// TIA Portal V21 export
FUNCTION "DELTA" : Void   // FC18, LAD
{ S7_Optimized_Access := 'TRUE' }
// stored: SetENOAutomatically false
   VAR_TEMP
      "F1 VALUE" : Real;
      "F2 VALUE" : Real;
      "F3 VALUE" : Real;
      "F4 VALUE" : Real;
      "F5 VALUE" : Real;
   END_VAR
   VAR_TEMP   // added for the SCL form of the ladder/FBD networks
      _w1 : Bool;
      _w2 : Bool;
      _w3 : Bool;
      _w4 : Bool;
      _w5 : Bool;
      _w6 : Bool;
      _w7 : Bool;
      _w8 : Bool;
      _w9 : Bool;
      _w10 : Bool;
      _w11 : Bool;
      _w12 : Bool;
   END_VAR
BEGIN

REGION Network 1
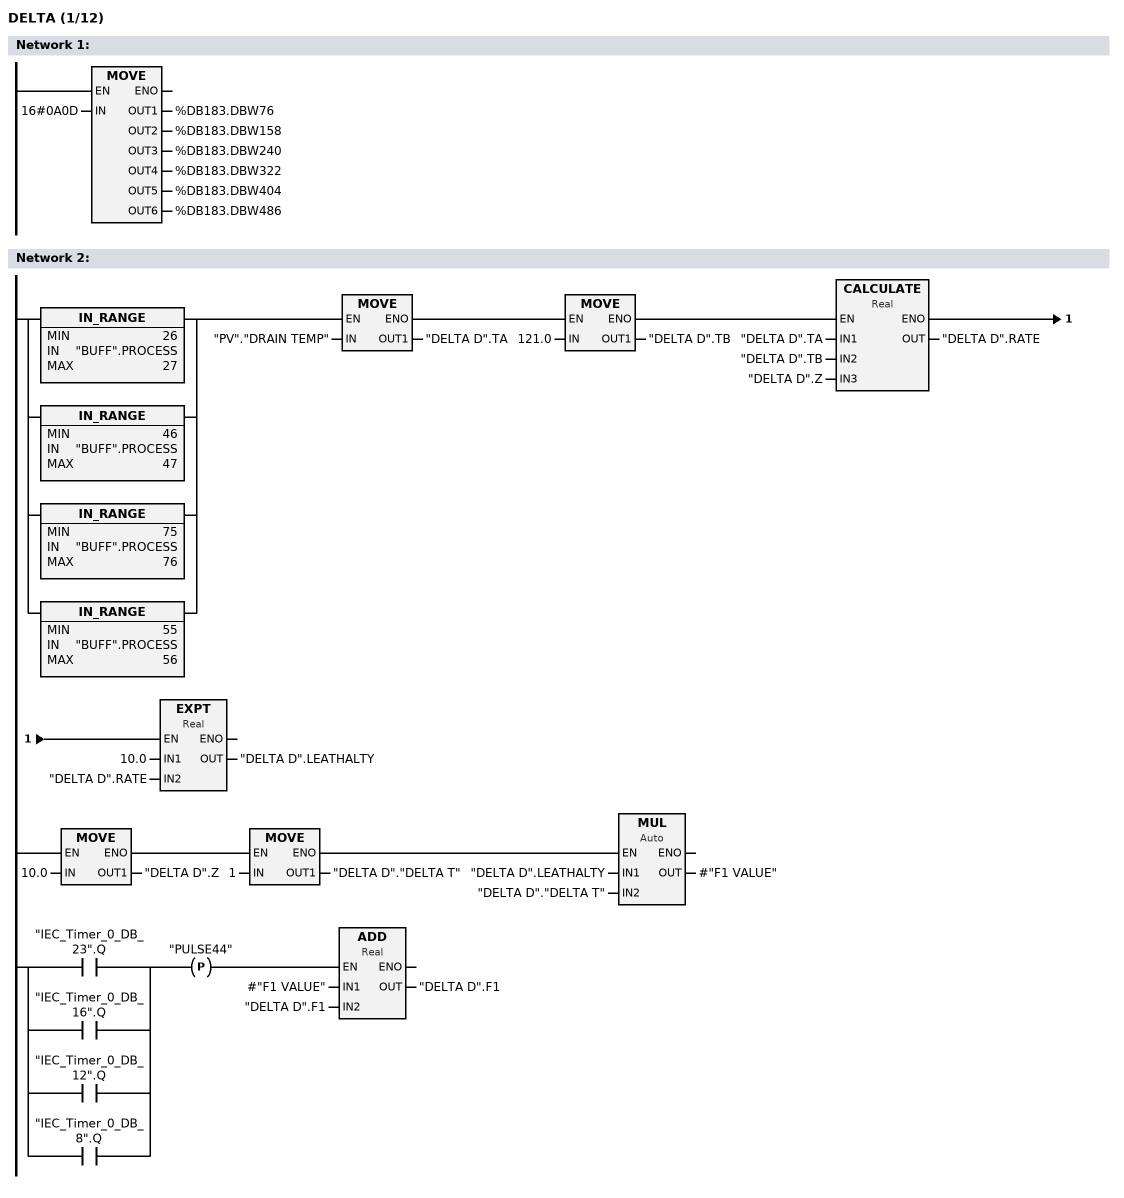
   RUNG wire#powerrail
      Move(in := 16#0A0D, out1 => %DB183.DBW76, out2 => %DB183.DBW158, out3 => %DB183.DBW240, out4 => %DB183.DBW322, out5 => %DB183.DBW404, out6 => %DB183.DBW486)
   END_RUNG
   // the same network as SCL:
   %DB183.DBW76 := 16#0A0D;
   %DB183.DBW158 := 16#0A0D;
   %DB183.DBW240 := 16#0A0D;
   %DB183.DBW322 := 16#0A0D;
   %DB183.DBW404 := 16#0A0D;
   %DB183.DBW486 := 16#0A0D;
END_REGION

REGION Network 2
   IF ((26 <= "BUFF".PROCESS) AND ("BUFF".PROCESS <= 27)) OR ((46 <= "BUFF".PROCESS) AND ("BUFF".PROCESS <= 47)) OR ((75 <= "BUFF".PROCESS) AND ("BUFF".PROCESS <= 76)) OR ((55 <= "BUFF".PROCESS) AND ("BUFF".PROCESS <= 56)) THEN
       "DELTA D".TA := "PV"."DRAIN TEMP";
       "DELTA D".TB := 121.0;
       "DELTA D".RATE := ("DELTA D".TA-"DELTA D".TB)/"DELTA D".Z;
       "DELTA D".LEATHALTY := 10.0 ** "DELTA D".RATE;
   END_IF;
   "DELTA D".Z := 10.0;
   "DELTA D"."DELTA T" := 1;
   #"F1 VALUE" := "DELTA D".LEATHALTY * "DELTA D"."DELTA T";
   #_w1 := "IEC_Timer_0_DB_23".Q OR "IEC_Timer_0_DB_16".Q OR "IEC_Timer_0_DB_12".Q OR "IEC_Timer_0_DB_8".Q;
   #_w2 := #_w1 AND NOT "PULSE44";   // rising edge
   "PULSE44" := #_w1;
   IF #_w2 THEN "DELTA D".F1 := #"F1 VALUE" + "DELTA D".F1; END_IF;
END_REGION

REGION Network 3
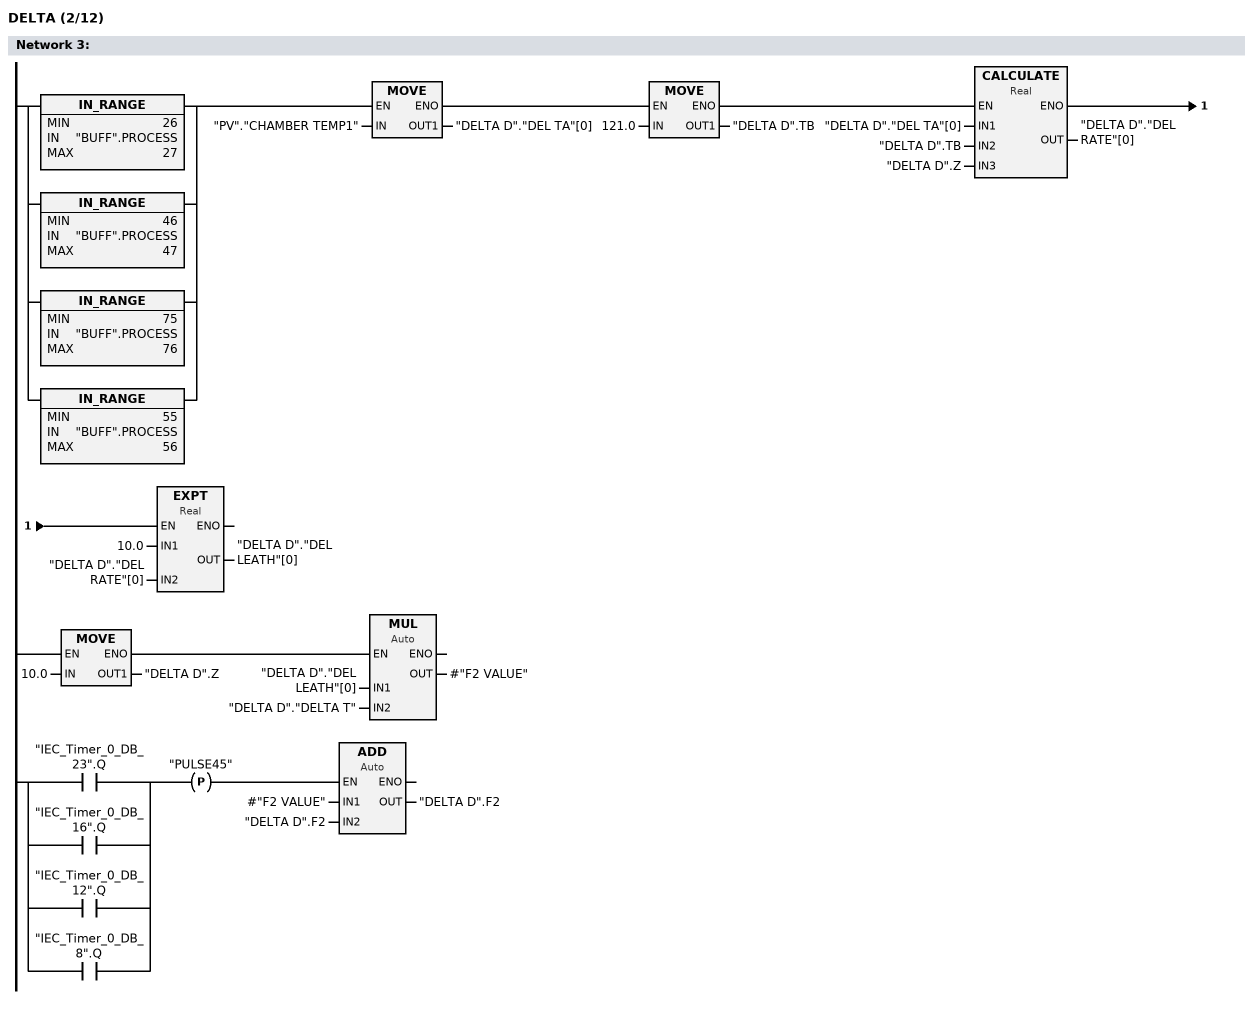
   IF ((26 <= "BUFF".PROCESS) AND ("BUFF".PROCESS <= 27)) OR ((46 <= "BUFF".PROCESS) AND ("BUFF".PROCESS <= 47)) OR ((75 <= "BUFF".PROCESS) AND ("BUFF".PROCESS <= 76)) OR ((55 <= "BUFF".PROCESS) AND ("BUFF".PROCESS <= 56)) THEN
       "DELTA D"."DEL TA"[0] := "PV"."CHAMBER TEMP1";
       "DELTA D".TB := 121.0;
       "DELTA D"."DEL RATE"[0] := ("DELTA D"."DEL TA"[0]-"DELTA D".TB)/"DELTA D".Z;
       "DELTA D"."DEL LEATH"[0] := 10.0 ** "DELTA D"."DEL RATE"[0];
   END_IF;
   "DELTA D".Z := 10.0;
   #"F2 VALUE" := "DELTA D"."DEL LEATH"[0] * "DELTA D"."DELTA T";
   #_w1 := "IEC_Timer_0_DB_23".Q OR "IEC_Timer_0_DB_16".Q OR "IEC_Timer_0_DB_12".Q OR "IEC_Timer_0_DB_8".Q;
   #_w2 := #_w1 AND NOT "PULSE45";   // rising edge
   "PULSE45" := #_w1;
   IF #_w2 THEN "DELTA D".F2 := #"F2 VALUE" + "DELTA D".F2; END_IF;
END_REGION

REGION Network 4
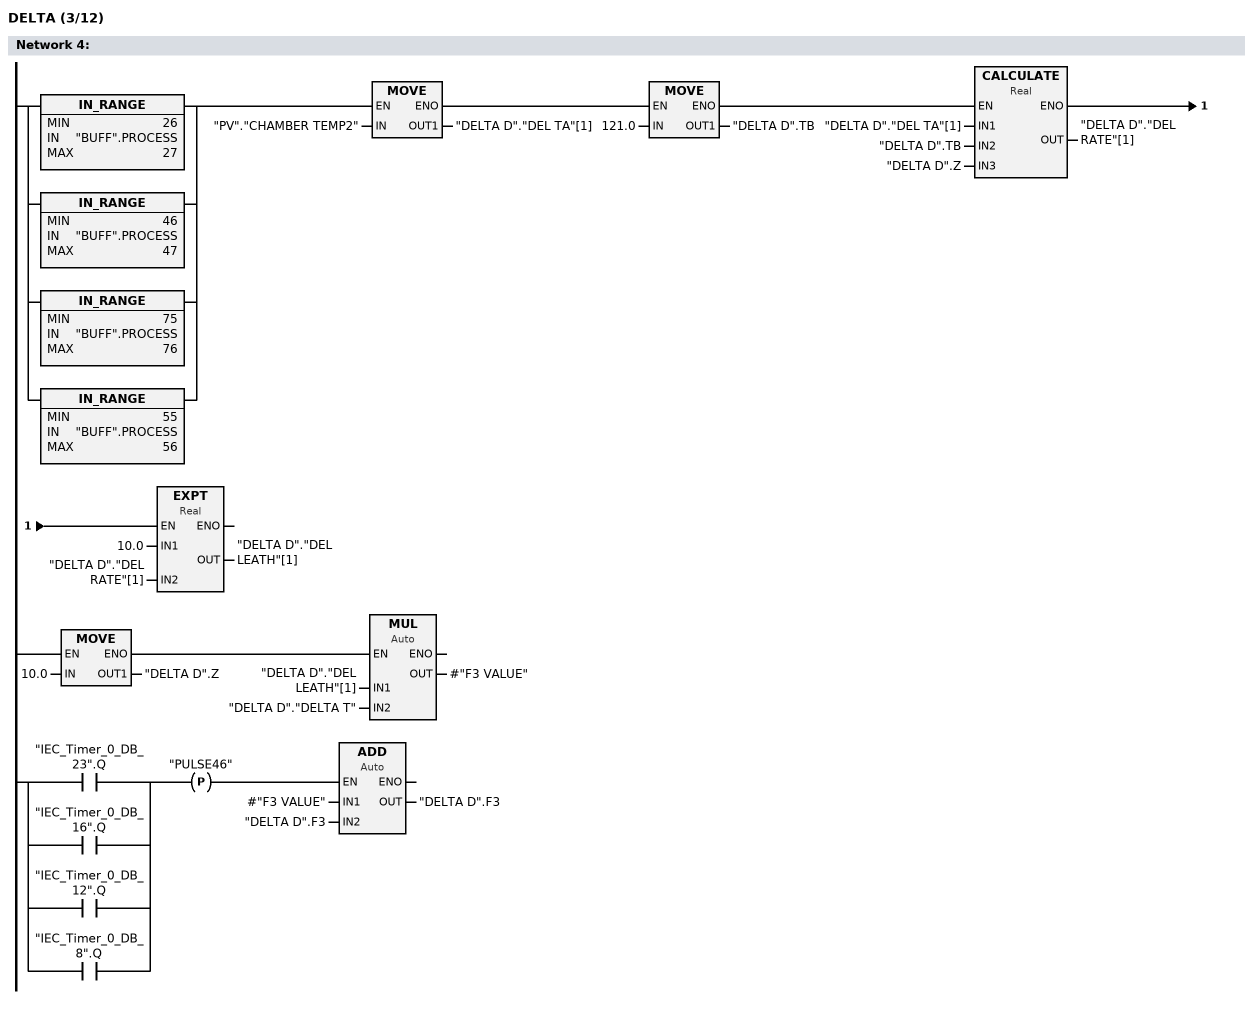
   IF ((26 <= "BUFF".PROCESS) AND ("BUFF".PROCESS <= 27)) OR ((46 <= "BUFF".PROCESS) AND ("BUFF".PROCESS <= 47)) OR ((75 <= "BUFF".PROCESS) AND ("BUFF".PROCESS <= 76)) OR ((55 <= "BUFF".PROCESS) AND ("BUFF".PROCESS <= 56)) THEN
       "DELTA D"."DEL TA"[1] := "PV"."CHAMBER TEMP2";
       "DELTA D".TB := 121.0;
       "DELTA D"."DEL RATE"[1] := ("DELTA D"."DEL TA"[1]-"DELTA D".TB)/"DELTA D".Z;
       "DELTA D"."DEL LEATH"[1] := 10.0 ** "DELTA D"."DEL RATE"[1];
   END_IF;
   "DELTA D".Z := 10.0;
   #"F3 VALUE" := "DELTA D"."DEL LEATH"[1] * "DELTA D"."DELTA T";
   #_w1 := "IEC_Timer_0_DB_23".Q OR "IEC_Timer_0_DB_16".Q OR "IEC_Timer_0_DB_12".Q OR "IEC_Timer_0_DB_8".Q;
   #_w2 := #_w1 AND NOT "PULSE46";   // rising edge
   "PULSE46" := #_w1;
   IF #_w2 THEN "DELTA D".F3 := #"F3 VALUE" + "DELTA D".F3; END_IF;
END_REGION

REGION Network 5
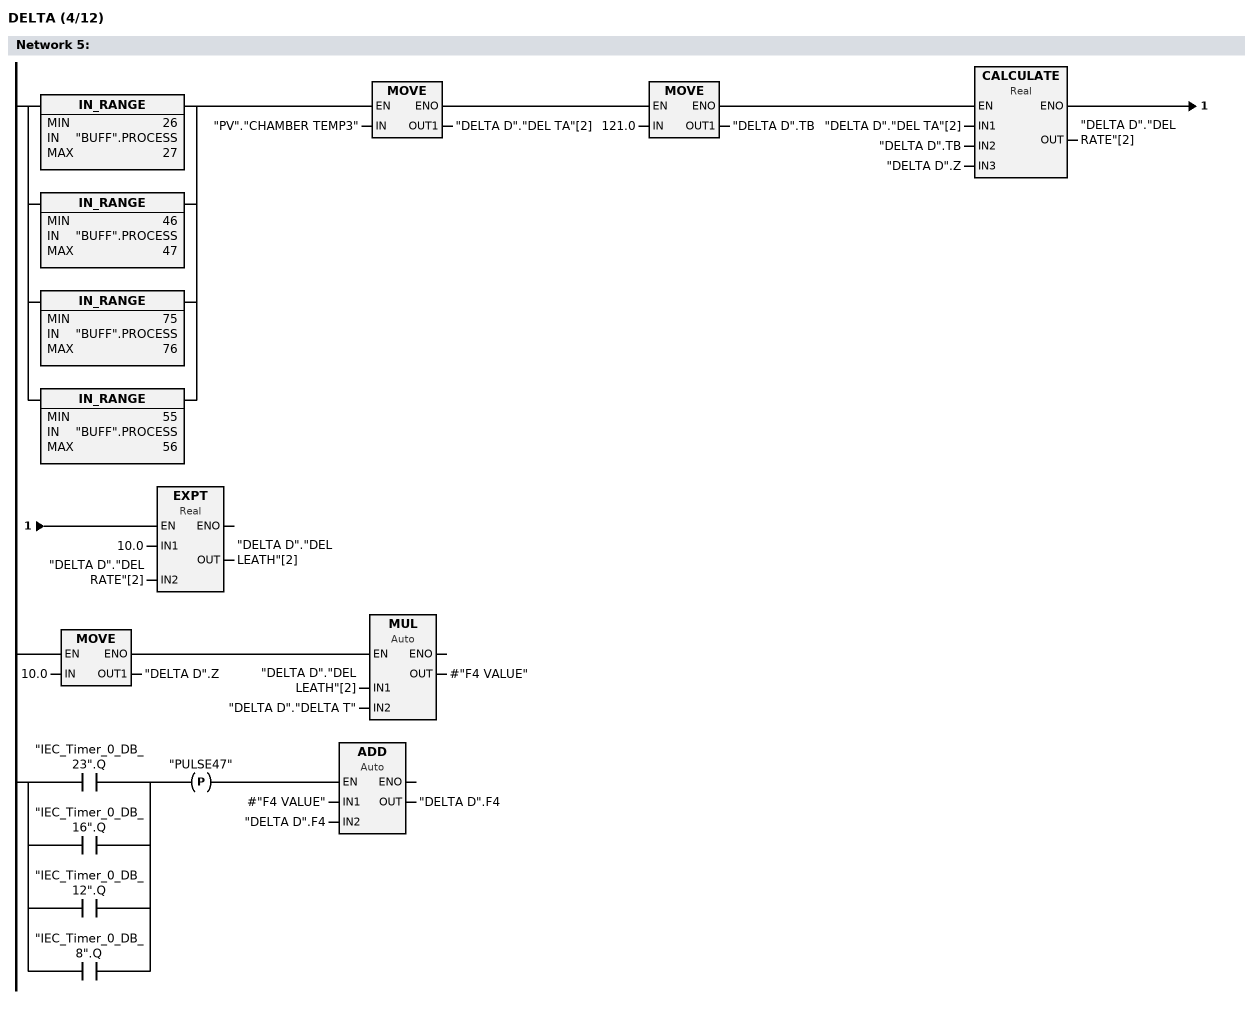
   IF ((26 <= "BUFF".PROCESS) AND ("BUFF".PROCESS <= 27)) OR ((46 <= "BUFF".PROCESS) AND ("BUFF".PROCESS <= 47)) OR ((75 <= "BUFF".PROCESS) AND ("BUFF".PROCESS <= 76)) OR ((55 <= "BUFF".PROCESS) AND ("BUFF".PROCESS <= 56)) THEN
       "DELTA D"."DEL TA"[2] := "PV"."CHAMBER TEMP3";
       "DELTA D".TB := 121.0;
       "DELTA D"."DEL RATE"[2] := ("DELTA D"."DEL TA"[2]-"DELTA D".TB)/"DELTA D".Z;
       "DELTA D"."DEL LEATH"[2] := 10.0 ** "DELTA D"."DEL RATE"[2];
   END_IF;
   "DELTA D".Z := 10.0;
   #"F4 VALUE" := "DELTA D"."DEL LEATH"[2] * "DELTA D"."DELTA T";
   #_w1 := "IEC_Timer_0_DB_23".Q OR "IEC_Timer_0_DB_16".Q OR "IEC_Timer_0_DB_12".Q OR "IEC_Timer_0_DB_8".Q;
   #_w2 := #_w1 AND NOT "PULSE47";   // rising edge
   "PULSE47" := #_w1;
   IF #_w2 THEN "DELTA D".F4 := #"F4 VALUE" + "DELTA D".F4; END_IF;
END_REGION

REGION Network 6
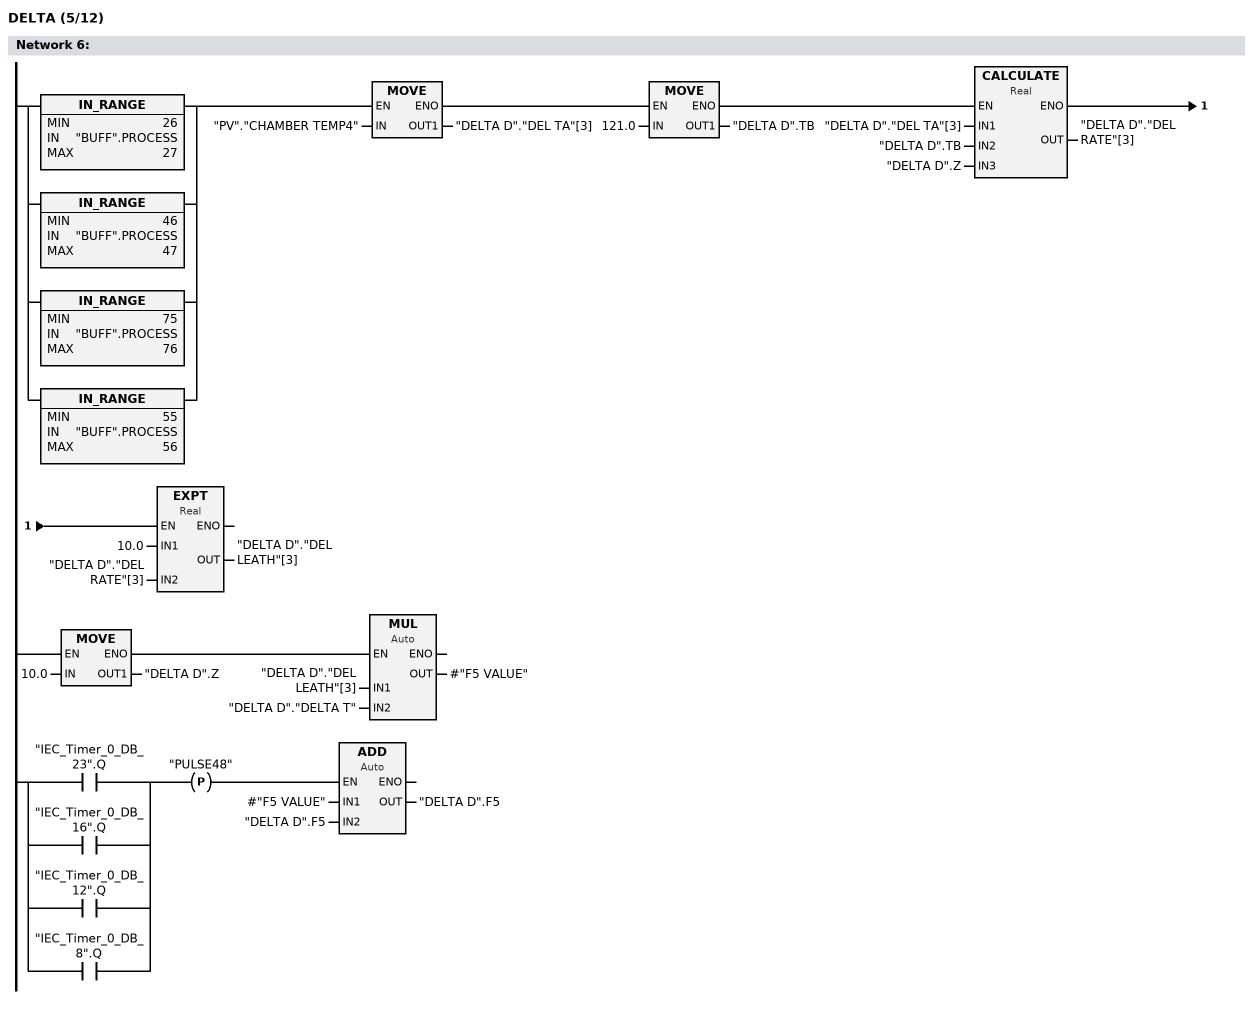
   IF ((26 <= "BUFF".PROCESS) AND ("BUFF".PROCESS <= 27)) OR ((46 <= "BUFF".PROCESS) AND ("BUFF".PROCESS <= 47)) OR ((75 <= "BUFF".PROCESS) AND ("BUFF".PROCESS <= 76)) OR ((55 <= "BUFF".PROCESS) AND ("BUFF".PROCESS <= 56)) THEN
       "DELTA D"."DEL TA"[3] := "PV"."CHAMBER TEMP4";
       "DELTA D".TB := 121.0;
       "DELTA D"."DEL RATE"[3] := ("DELTA D"."DEL TA"[3]-"DELTA D".TB)/"DELTA D".Z;
       "DELTA D"."DEL LEATH"[3] := 10.0 ** "DELTA D"."DEL RATE"[3];
   END_IF;
   "DELTA D".Z := 10.0;
   #"F5 VALUE" := "DELTA D"."DEL LEATH"[3] * "DELTA D"."DELTA T";
   #_w1 := "IEC_Timer_0_DB_23".Q OR "IEC_Timer_0_DB_16".Q OR "IEC_Timer_0_DB_12".Q OR "IEC_Timer_0_DB_8".Q;
   #_w2 := #_w1 AND NOT "PULSE48";   // rising edge
   "PULSE48" := #_w1;
   IF #_w2 THEN "DELTA D".F5 := #"F5 VALUE" + "DELTA D".F5; END_IF;
END_REGION

REGION Network 7
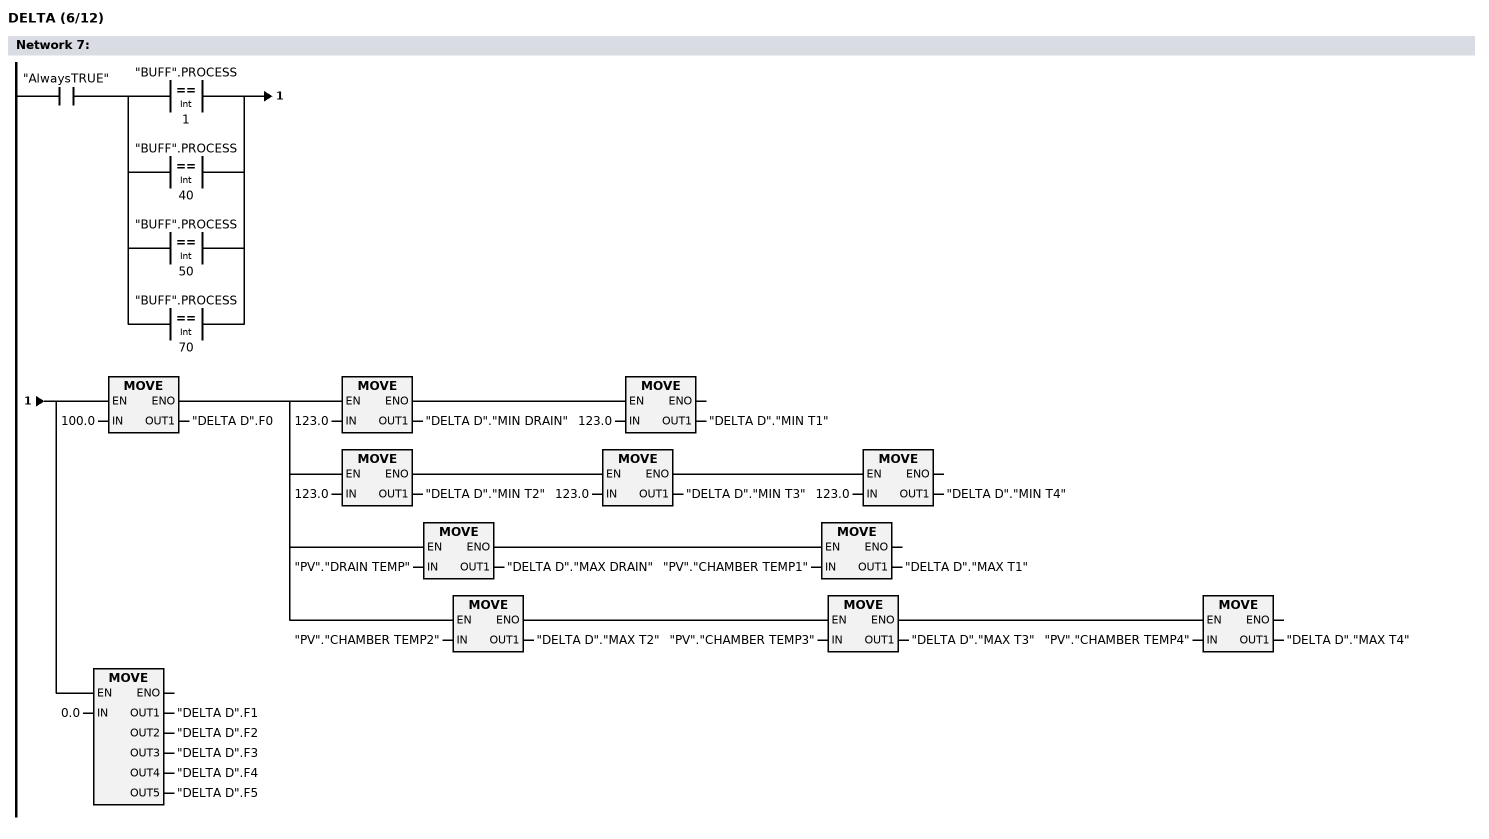
   RUNG wire#powerrail
      Contact( "AlwaysTRUE" )
      wire#w1
      { S7_Templates := "SrcType := Int" } EQ_Contact(in1 := "BUFF".PROCESS, in2 := 1)
      wire#w2
      Move(in := 100.0, out1 => "DELTA D".F0)
      wire#w3
      Move(in := 123.0, out1 => "DELTA D"."MIN DRAIN")
      Move(in := 123.0, out1 => "DELTA D"."MIN T1")
   END_RUNG
   RUNG wire#w1
      { S7_Templates := "SrcType := Int" } EQ_Contact(in1 := "BUFF".PROCESS, in2 := 40)
   END_RUNG wire#w2
   RUNG wire#w1
      { S7_Templates := "SrcType := Int" } EQ_Contact(in1 := "BUFF".PROCESS, in2 := 50)
   END_RUNG wire#w2
   RUNG wire#w1
      { S7_Templates := "SrcType := Int" } EQ_Contact(in1 := "BUFF".PROCESS, in2 := 70)
   END_RUNG wire#w2
   RUNG wire#w3
      Move(in := 123.0, out1 => "DELTA D"."MIN T2")
      Move(in := 123.0, out1 => "DELTA D"."MIN T3")
      Move(in := 123.0, out1 => "DELTA D"."MIN T4")
   END_RUNG
   RUNG wire#w3
      Move(in := "PV"."DRAIN TEMP", out1 => "DELTA D"."MAX DRAIN")
      Move(in := "PV"."CHAMBER TEMP1", out1 => "DELTA D"."MAX T1")
   END_RUNG
   RUNG wire#w3
      Move(in := "PV"."CHAMBER TEMP2", out1 => "DELTA D"."MAX T2")
      Move(in := "PV"."CHAMBER TEMP3", out1 => "DELTA D"."MAX T3")
      Move(in := "PV"."CHAMBER TEMP4", out1 => "DELTA D"."MAX T4")
   END_RUNG
   RUNG wire#w2
      Move(in := 0.0, out1 => "DELTA D".F1, out2 => "DELTA D".F2, out3 => "DELTA D".F3, out4 => "DELTA D".F4, out5 => "DELTA D".F5)
   END_RUNG
   // the same network as SCL:
   IF "AlwaysTRUE" AND (("BUFF".PROCESS = 1) OR ("BUFF".PROCESS = 40) OR ("BUFF".PROCESS = 50) OR ("BUFF".PROCESS = 70)) THEN
       "DELTA D".F0 := 100.0;
       "DELTA D"."MIN DRAIN" := 123.0;
       "DELTA D"."MIN T1" := 123.0;
       "DELTA D"."MIN T2" := 123.0;
       "DELTA D"."MIN T3" := 123.0;
       "DELTA D"."MIN T4" := 123.0;
       "DELTA D"."MAX DRAIN" := "PV"."DRAIN TEMP";
       "DELTA D"."MAX T1" := "PV"."CHAMBER TEMP1";
       "DELTA D"."MAX T2" := "PV"."CHAMBER TEMP2";
       "DELTA D"."MAX T3" := "PV"."CHAMBER TEMP3";
       "DELTA D"."MAX T4" := "PV"."CHAMBER TEMP4";
       "DELTA D".F1 := 0.0;
       "DELTA D".F2 := 0.0;
       "DELTA D".F3 := 0.0;
       "DELTA D".F4 := 0.0;
       "DELTA D".F5 := 0.0;
   END_IF;
END_REGION

REGION Network 8
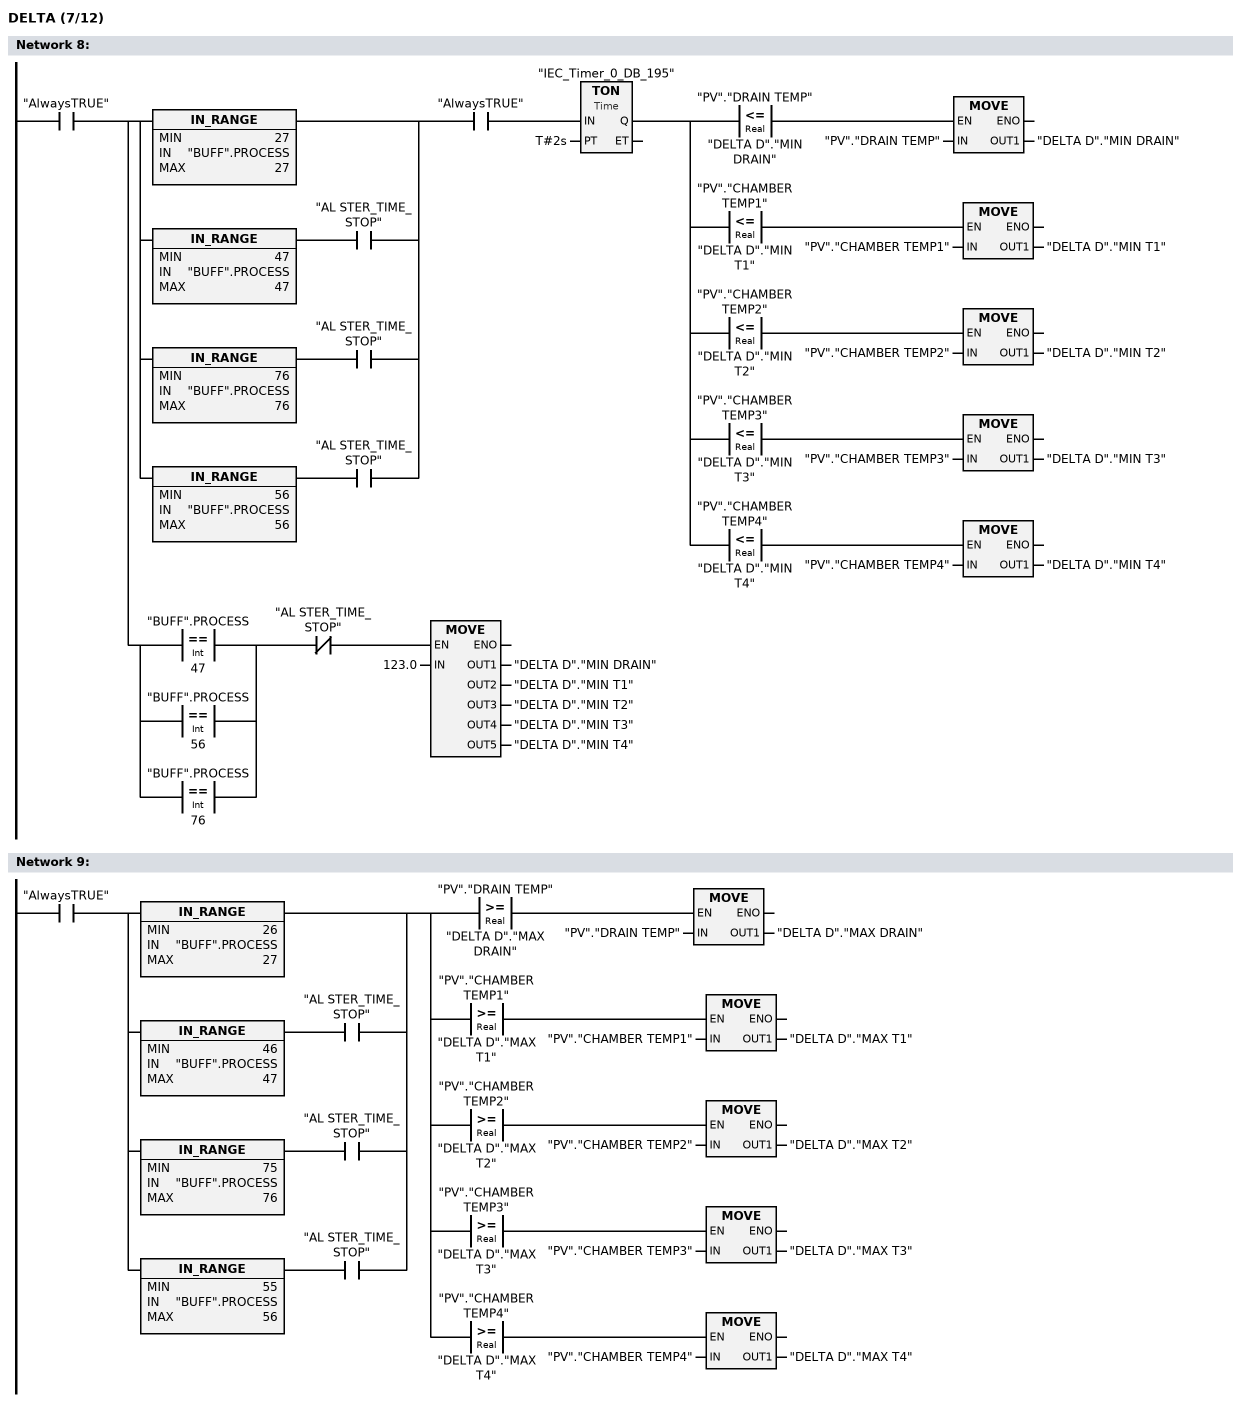
   RUNG wire#powerrail
      Contact( "AlwaysTRUE" )
      wire#w1
      { S7_Templates := "SrcType := Int" } InRange(min := 27, in := "BUFF".PROCESS, max := 27)
      wire#w2
      Contact( "AlwaysTRUE" )
      { S7_Templates := "time_type := Time" } "IEC_Timer_0_DB_195".TON(pt := T#2s, et =>)
      wire#w3
      { S7_Templates := "SrcType := Real" } LE_Contact(in1 := "PV"."DRAIN TEMP", in2 := "DELTA D"."MIN DRAIN")
      Move(in := "PV"."DRAIN TEMP", out1 => "DELTA D"."MIN DRAIN")
   END_RUNG
   RUNG wire#w1
      { S7_Templates := "SrcType := Int" } InRange(min := 47, in := "BUFF".PROCESS, max := 47)
      Contact( "AL STER_TIME_STOP" )
   END_RUNG wire#w2
   RUNG wire#w1
      { S7_Templates := "SrcType := Int" } InRange(min := 76, in := "BUFF".PROCESS, max := 76)
      Contact( "AL STER_TIME_STOP" )
   END_RUNG wire#w2
   RUNG wire#w1
      { S7_Templates := "SrcType := Int" } InRange(min := 56, in := "BUFF".PROCESS, max := 56)
      Contact( "AL STER_TIME_STOP" )
   END_RUNG wire#w2
   RUNG wire#w3
      { S7_Templates := "SrcType := Real" } LE_Contact(in1 := "PV"."CHAMBER TEMP1", in2 := "DELTA D"."MIN T1")
      Move(in := "PV"."CHAMBER TEMP1", out1 => "DELTA D"."MIN T1")
   END_RUNG
   RUNG wire#w3
      { S7_Templates := "SrcType := Real" } LE_Contact(in1 := "PV"."CHAMBER TEMP2", in2 := "DELTA D"."MIN T2")
      Move(in := "PV"."CHAMBER TEMP2", out1 => "DELTA D"."MIN T2")
   END_RUNG
   RUNG wire#w3
      { S7_Templates := "SrcType := Real" } LE_Contact(in1 := "PV"."CHAMBER TEMP3", in2 := "DELTA D"."MIN T3")
      Move(in := "PV"."CHAMBER TEMP3", out1 => "DELTA D"."MIN T3")
   END_RUNG
   RUNG wire#w3
      { S7_Templates := "SrcType := Real" } LE_Contact(in1 := "PV"."CHAMBER TEMP4", in2 := "DELTA D"."MIN T4")
      Move(in := "PV"."CHAMBER TEMP4", out1 => "DELTA D"."MIN T4")
   END_RUNG
   RUNG wire#w1
      { S7_Templates := "SrcType := Int" } EQ_Contact(in1 := "BUFF".PROCESS, in2 := 47)
      wire#w4
      I_Contact( "AL STER_TIME_STOP" )
      Move(in := 123.0, out1 => "DELTA D"."MIN DRAIN", out2 => "DELTA D"."MIN T1", out3 => "DELTA D"."MIN T2", out4 => "DELTA D"."MIN T3", out5 => "DELTA D"."MIN T4")
   END_RUNG
   RUNG wire#w1
      { S7_Templates := "SrcType := Int" } EQ_Contact(in1 := "BUFF".PROCESS, in2 := 56)
   END_RUNG wire#w4
   RUNG wire#w1
      { S7_Templates := "SrcType := Int" } EQ_Contact(in1 := "BUFF".PROCESS, in2 := 76)
   END_RUNG wire#w4
   // the same network as SCL:
   "IEC_Timer_0_DB_195".TON(IN := "AlwaysTRUE" AND (((27 <= "BUFF".PROCESS) AND ("BUFF".PROCESS <= 27)) OR ((47 <= "BUFF".PROCESS) AND ("BUFF".PROCESS <= 47) AND "AL STER_TIME_STOP") OR ((76 <= "BUFF".PROCESS) AND ("BUFF".PROCESS <= 76) AND "AL STER_TIME_STOP") OR ((56 <= "BUFF".PROCESS) AND ("BUFF".PROCESS <= 56) AND "AL STER_TIME_STOP")) AND "AlwaysTRUE",
                           PT := T#2s);
   IF "IEC_Timer_0_DB_195".Q AND ("PV"."DRAIN TEMP" <= "DELTA D"."MIN DRAIN") THEN
       "DELTA D"."MIN DRAIN" := "PV"."DRAIN TEMP";
   END_IF;
   IF "IEC_Timer_0_DB_195".Q AND ("PV"."CHAMBER TEMP1" <= "DELTA D"."MIN T1") THEN
       "DELTA D"."MIN T1" := "PV"."CHAMBER TEMP1";
   END_IF;
   IF "IEC_Timer_0_DB_195".Q AND ("PV"."CHAMBER TEMP2" <= "DELTA D"."MIN T2") THEN
       "DELTA D"."MIN T2" := "PV"."CHAMBER TEMP2";
   END_IF;
   IF "IEC_Timer_0_DB_195".Q AND ("PV"."CHAMBER TEMP3" <= "DELTA D"."MIN T3") THEN
       "DELTA D"."MIN T3" := "PV"."CHAMBER TEMP3";
   END_IF;
   IF "IEC_Timer_0_DB_195".Q AND ("PV"."CHAMBER TEMP4" <= "DELTA D"."MIN T4") THEN
       "DELTA D"."MIN T4" := "PV"."CHAMBER TEMP4";
   END_IF;
   IF "AlwaysTRUE" AND (("BUFF".PROCESS = 47) OR ("BUFF".PROCESS = 56) OR ("BUFF".PROCESS = 76)) AND NOT "AL STER_TIME_STOP" THEN
       "DELTA D"."MIN DRAIN" := 123.0;
       "DELTA D"."MIN T1" := 123.0;
       "DELTA D"."MIN T2" := 123.0;
       "DELTA D"."MIN T3" := 123.0;
       "DELTA D"."MIN T4" := 123.0;
   END_IF;
END_REGION

REGION Network 9
   RUNG wire#powerrail
      Contact( "AlwaysTRUE" )
      wire#w1
      { S7_Templates := "SrcType := Int" } InRange(min := 26, in := "BUFF".PROCESS, max := 27)
      wire#w2
      { S7_Templates := "SrcType := Real" } GE_Contact(in1 := "PV"."DRAIN TEMP", in2 := "DELTA D"."MAX DRAIN")
      Move(in := "PV"."DRAIN TEMP", out1 => "DELTA D"."MAX DRAIN")
   END_RUNG
   RUNG wire#w1
      { S7_Templates := "SrcType := Int" } InRange(min := 46, in := "BUFF".PROCESS, max := 47)
      Contact( "AL STER_TIME_STOP" )
   END_RUNG wire#w2
   RUNG wire#w1
      { S7_Templates := "SrcType := Int" } InRange(min := 75, in := "BUFF".PROCESS, max := 76)
      Contact( "AL STER_TIME_STOP" )
   END_RUNG wire#w2
   RUNG wire#w1
      { S7_Templates := "SrcType := Int" } InRange(min := 55, in := "BUFF".PROCESS, max := 56)
      Contact( "AL STER_TIME_STOP" )
   END_RUNG wire#w2
   RUNG wire#w2
      { S7_Templates := "SrcType := Real" } GE_Contact(in1 := "PV"."CHAMBER TEMP1", in2 := "DELTA D"."MAX T1")
      Move(in := "PV"."CHAMBER TEMP1", out1 => "DELTA D"."MAX T1")
   END_RUNG
   RUNG wire#w2
      { S7_Templates := "SrcType := Real" } GE_Contact(in1 := "PV"."CHAMBER TEMP2", in2 := "DELTA D"."MAX T2")
      Move(in := "PV"."CHAMBER TEMP2", out1 => "DELTA D"."MAX T2")
   END_RUNG
   RUNG wire#w2
      { S7_Templates := "SrcType := Real" } GE_Contact(in1 := "PV"."CHAMBER TEMP3", in2 := "DELTA D"."MAX T3")
      Move(in := "PV"."CHAMBER TEMP3", out1 => "DELTA D"."MAX T3")
   END_RUNG
   RUNG wire#w2
      { S7_Templates := "SrcType := Real" } GE_Contact(in1 := "PV"."CHAMBER TEMP4", in2 := "DELTA D"."MAX T4")
      Move(in := "PV"."CHAMBER TEMP4", out1 => "DELTA D"."MAX T4")
   END_RUNG
   // the same network as SCL:
   #_w1 := "AlwaysTRUE" AND (((26 <= "BUFF".PROCESS) AND ("BUFF".PROCESS <= 27)) OR ((46 <= "BUFF".PROCESS) AND ("BUFF".PROCESS <= 47) AND "AL STER_TIME_STOP") OR ((75 <= "BUFF".PROCESS) AND ("BUFF".PROCESS <= 76) AND "AL STER_TIME_STOP") OR ((55 <= "BUFF".PROCESS) AND ("BUFF".PROCESS <= 56) AND "AL STER_TIME_STOP"));
   IF #_w1 AND ("PV"."DRAIN TEMP" >= "DELTA D"."MAX DRAIN") THEN
       "DELTA D"."MAX DRAIN" := "PV"."DRAIN TEMP";
   END_IF;
   IF #_w1 AND ("PV"."CHAMBER TEMP1" >= "DELTA D"."MAX T1") THEN
       "DELTA D"."MAX T1" := "PV"."CHAMBER TEMP1";
   END_IF;
   IF #_w1 AND ("PV"."CHAMBER TEMP2" >= "DELTA D"."MAX T2") THEN
       "DELTA D"."MAX T2" := "PV"."CHAMBER TEMP2";
   END_IF;
   IF #_w1 AND ("PV"."CHAMBER TEMP3" >= "DELTA D"."MAX T3") THEN
       "DELTA D"."MAX T3" := "PV"."CHAMBER TEMP3";
   END_IF;
   IF #_w1 AND ("PV"."CHAMBER TEMP4" >= "DELTA D"."MAX T4") THEN
       "DELTA D"."MAX T4" := "PV"."CHAMBER TEMP4";
   END_IF;
END_REGION

REGION Network 10
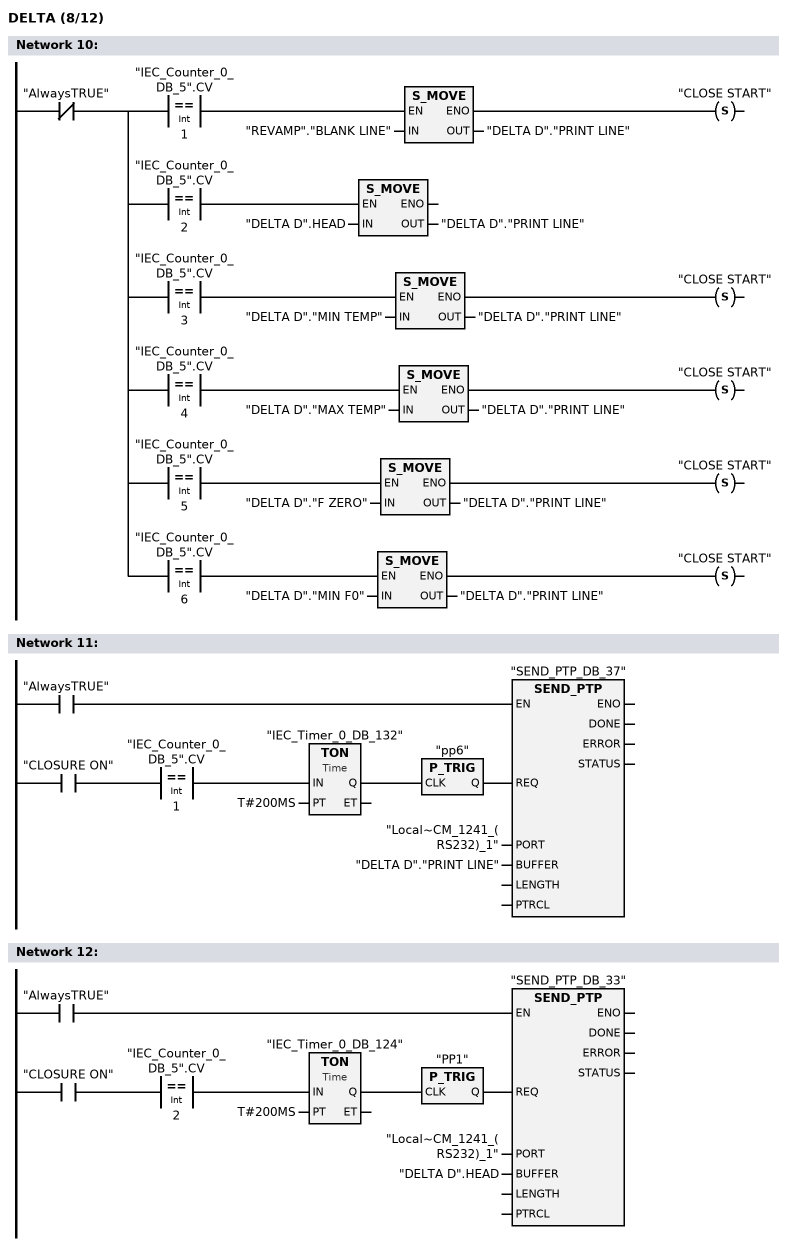
   RUNG wire#powerrail
      I_Contact( "AlwaysTRUE" )
      wire#w1
      { S7_Templates := "SrcType := Int" } EQ_Contact(in1 := "IEC_Counter_0_DB_5".CV, in2 := 1)
      S_Move(in := "REVAMP"."BLANK LINE", out => "DELTA D"."PRINT LINE")
      S_Coil( "CLOSE START" )
   END_RUNG
   RUNG wire#w1
      { S7_Templates := "SrcType := Int" } EQ_Contact(in1 := "IEC_Counter_0_DB_5".CV, in2 := 2)
      S_Move(in := "DELTA D".HEAD, out => "DELTA D"."PRINT LINE")
   END_RUNG
   RUNG wire#w1
      { S7_Templates := "SrcType := Int" } EQ_Contact(in1 := "IEC_Counter_0_DB_5".CV, in2 := 3)
      S_Move(in := "DELTA D"."MIN TEMP", out => "DELTA D"."PRINT LINE")
      S_Coil( "CLOSE START" )
   END_RUNG
   RUNG wire#w1
      { S7_Templates := "SrcType := Int" } EQ_Contact(in1 := "IEC_Counter_0_DB_5".CV, in2 := 4)
      S_Move(in := "DELTA D"."MAX TEMP", out => "DELTA D"."PRINT LINE")
      S_Coil( "CLOSE START" )
   END_RUNG
   RUNG wire#w1
      { S7_Templates := "SrcType := Int" } EQ_Contact(in1 := "IEC_Counter_0_DB_5".CV, in2 := 5)
      S_Move(in := "DELTA D"."F ZERO", out => "DELTA D"."PRINT LINE")
      S_Coil( "CLOSE START" )
   END_RUNG
   RUNG wire#w1
      { S7_Templates := "SrcType := Int" } EQ_Contact(in1 := "IEC_Counter_0_DB_5".CV, in2 := 6)
      S_Move(in := "DELTA D"."MIN F0", out => "DELTA D"."PRINT LINE")
      S_Coil( "CLOSE START" )
   END_RUNG
   // the same network as SCL:
   IF NOT "AlwaysTRUE" AND ("IEC_Counter_0_DB_5".CV = 1) THEN
       "DELTA D"."PRINT LINE" := "REVAMP"."BLANK LINE";
       "CLOSE START" := TRUE;
   END_IF;
   IF NOT "AlwaysTRUE" AND ("IEC_Counter_0_DB_5".CV = 2) THEN
       "DELTA D"."PRINT LINE" := "DELTA D".HEAD;
   END_IF;
   IF NOT "AlwaysTRUE" AND ("IEC_Counter_0_DB_5".CV = 3) THEN
       "DELTA D"."PRINT LINE" := "DELTA D"."MIN TEMP";
       "CLOSE START" := TRUE;
   END_IF;
   IF NOT "AlwaysTRUE" AND ("IEC_Counter_0_DB_5".CV = 4) THEN
       "DELTA D"."PRINT LINE" := "DELTA D"."MAX TEMP";
       "CLOSE START" := TRUE;
   END_IF;
   IF NOT "AlwaysTRUE" AND ("IEC_Counter_0_DB_5".CV = 5) THEN
       "DELTA D"."PRINT LINE" := "DELTA D"."F ZERO";
       "CLOSE START" := TRUE;
   END_IF;
   IF NOT "AlwaysTRUE" AND ("IEC_Counter_0_DB_5".CV = 6) THEN
       "DELTA D"."PRINT LINE" := "DELTA D"."MIN F0";
       "CLOSE START" := TRUE;
   END_IF;
END_REGION

REGION Network 11
   RUNG wire#powerrail
      Contact( "AlwaysTRUE" )
      "SEND_PTP_DB_37".SEND_PTP(REQ := wire#w1, PORT := "Local~CM_1241_(RS232)_1", BUFFER := "DELTA D"."PRINT LINE", LENGTH :=, PTRCL :=, DONE =>, ERROR =>, STATUS =>)
   END_RUNG
   RUNG wire#powerrail
      Contact( "CLOSURE ON" )
      { S7_Templates := "SrcType := Int" } EQ_Contact(in1 := "IEC_Counter_0_DB_5".CV, in2 := 1)
      { S7_Templates := "time_type := Time" } "IEC_Timer_0_DB_132".TON(pt := T#200MS, et =>)
      P_Trig( "pp6" )
   END_RUNG wire#w1
   // the same network as SCL:
   "IEC_Timer_0_DB_132".TON(IN := "CLOSURE ON" AND ("IEC_Counter_0_DB_5".CV = 1), PT := T#200MS);
   #_w1 := "IEC_Timer_0_DB_132".Q AND NOT "pp6";   // rising edge
   "pp6" := "IEC_Timer_0_DB_132".Q;
   IF "AlwaysTRUE" THEN
       "SEND_PTP_DB_37"(REQ := #_w1, PORT := "Local~CM_1241_(RS232)_1", BUFFER := "DELTA D"."PRINT LINE");   // SEND_PTP
   END_IF;
END_REGION

REGION Network 12
   RUNG wire#powerrail
      Contact( "AlwaysTRUE" )
      "SEND_PTP_DB_33".SEND_PTP(REQ := wire#w1, PORT := "Local~CM_1241_(RS232)_1", BUFFER := "DELTA D".HEAD, LENGTH :=, PTRCL :=, DONE =>, ERROR =>, STATUS =>)
   END_RUNG
   RUNG wire#powerrail
      Contact( "CLOSURE ON" )
      { S7_Templates := "SrcType := Int" } EQ_Contact(in1 := "IEC_Counter_0_DB_5".CV, in2 := 2)
      { S7_Templates := "time_type := Time" } "IEC_Timer_0_DB_124".TON(pt := T#200MS, et =>)
      P_Trig( "PP1" )
   END_RUNG wire#w1
   // the same network as SCL:
   "IEC_Timer_0_DB_124".TON(IN := "CLOSURE ON" AND ("IEC_Counter_0_DB_5".CV = 2), PT := T#200MS);
   #_w1 := "IEC_Timer_0_DB_124".Q AND NOT "PP1";   // rising edge
   "PP1" := "IEC_Timer_0_DB_124".Q;
   IF "AlwaysTRUE" THEN
       "SEND_PTP_DB_33"(REQ := #_w1, PORT := "Local~CM_1241_(RS232)_1", BUFFER := "DELTA D".HEAD);   // SEND_PTP
   END_IF;
END_REGION

REGION Network 13
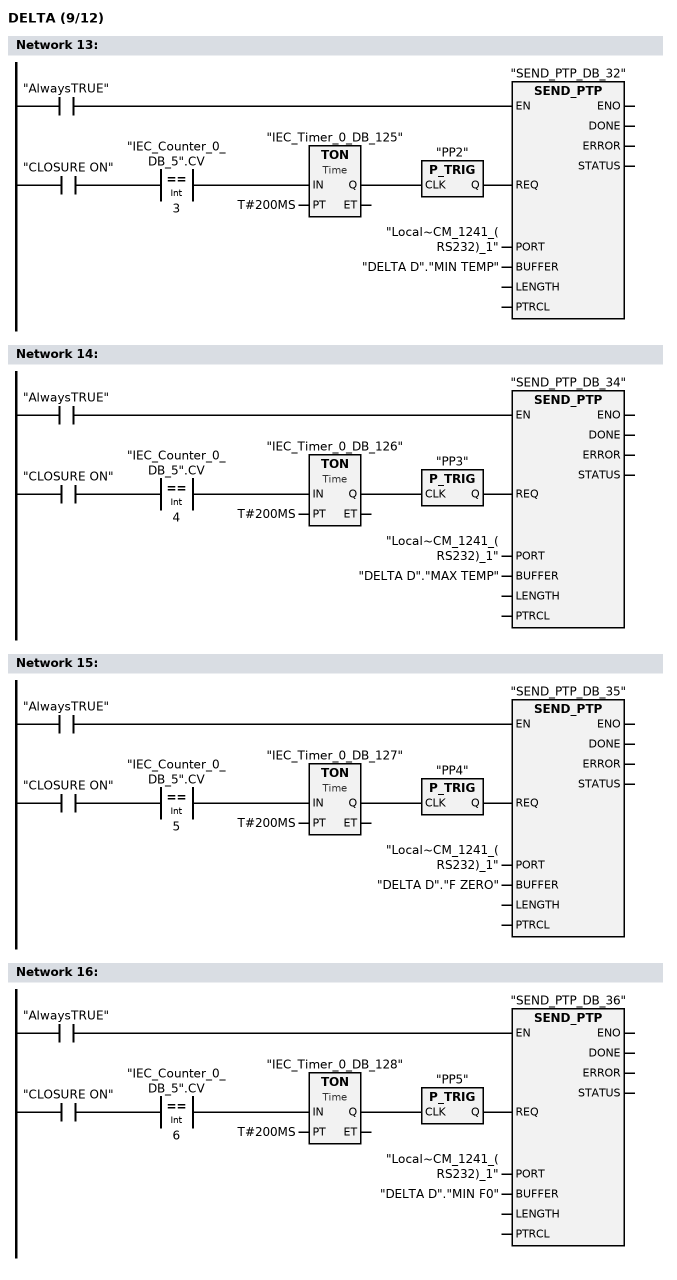
   RUNG wire#powerrail
      Contact( "AlwaysTRUE" )
      "SEND_PTP_DB_32".SEND_PTP(REQ := wire#w1, PORT := "Local~CM_1241_(RS232)_1", BUFFER := "DELTA D"."MIN TEMP", LENGTH :=, PTRCL :=, DONE =>, ERROR =>, STATUS =>)
   END_RUNG
   RUNG wire#powerrail
      Contact( "CLOSURE ON" )
      { S7_Templates := "SrcType := Int" } EQ_Contact(in1 := "IEC_Counter_0_DB_5".CV, in2 := 3)
      { S7_Templates := "time_type := Time" } "IEC_Timer_0_DB_125".TON(pt := T#200MS, et =>)
      P_Trig( "PP2" )
   END_RUNG wire#w1
   // the same network as SCL:
   "IEC_Timer_0_DB_125".TON(IN := "CLOSURE ON" AND ("IEC_Counter_0_DB_5".CV = 3), PT := T#200MS);
   #_w1 := "IEC_Timer_0_DB_125".Q AND NOT "PP2";   // rising edge
   "PP2" := "IEC_Timer_0_DB_125".Q;
   IF "AlwaysTRUE" THEN
       "SEND_PTP_DB_32"(REQ := #_w1, PORT := "Local~CM_1241_(RS232)_1", BUFFER := "DELTA D"."MIN TEMP");   // SEND_PTP
   END_IF;
END_REGION

REGION Network 14
   RUNG wire#powerrail
      Contact( "AlwaysTRUE" )
      "SEND_PTP_DB_34".SEND_PTP(REQ := wire#w1, PORT := "Local~CM_1241_(RS232)_1", BUFFER := "DELTA D"."MAX TEMP", LENGTH :=, PTRCL :=, DONE =>, ERROR =>, STATUS =>)
   END_RUNG
   RUNG wire#powerrail
      Contact( "CLOSURE ON" )
      { S7_Templates := "SrcType := Int" } EQ_Contact(in1 := "IEC_Counter_0_DB_5".CV, in2 := 4)
      { S7_Templates := "time_type := Time" } "IEC_Timer_0_DB_126".TON(pt := T#200MS, et =>)
      P_Trig( "PP3" )
   END_RUNG wire#w1
   // the same network as SCL:
   "IEC_Timer_0_DB_126".TON(IN := "CLOSURE ON" AND ("IEC_Counter_0_DB_5".CV = 4), PT := T#200MS);
   #_w1 := "IEC_Timer_0_DB_126".Q AND NOT "PP3";   // rising edge
   "PP3" := "IEC_Timer_0_DB_126".Q;
   IF "AlwaysTRUE" THEN
       "SEND_PTP_DB_34"(REQ := #_w1, PORT := "Local~CM_1241_(RS232)_1", BUFFER := "DELTA D"."MAX TEMP");   // SEND_PTP
   END_IF;
END_REGION

REGION Network 15
   RUNG wire#powerrail
      Contact( "AlwaysTRUE" )
      "SEND_PTP_DB_35".SEND_PTP(REQ := wire#w1, PORT := "Local~CM_1241_(RS232)_1", BUFFER := "DELTA D"."F ZERO", LENGTH :=, PTRCL :=, DONE =>, ERROR =>, STATUS =>)
   END_RUNG
   RUNG wire#powerrail
      Contact( "CLOSURE ON" )
      { S7_Templates := "SrcType := Int" } EQ_Contact(in1 := "IEC_Counter_0_DB_5".CV, in2 := 5)
      { S7_Templates := "time_type := Time" } "IEC_Timer_0_DB_127".TON(pt := T#200MS, et =>)
      P_Trig( "PP4" )
   END_RUNG wire#w1
   // the same network as SCL:
   "IEC_Timer_0_DB_127".TON(IN := "CLOSURE ON" AND ("IEC_Counter_0_DB_5".CV = 5), PT := T#200MS);
   #_w1 := "IEC_Timer_0_DB_127".Q AND NOT "PP4";   // rising edge
   "PP4" := "IEC_Timer_0_DB_127".Q;
   IF "AlwaysTRUE" THEN
       "SEND_PTP_DB_35"(REQ := #_w1, PORT := "Local~CM_1241_(RS232)_1", BUFFER := "DELTA D"."F ZERO");   // SEND_PTP
   END_IF;
END_REGION

REGION Network 16
   RUNG wire#powerrail
      Contact( "AlwaysTRUE" )
      "SEND_PTP_DB_36".SEND_PTP(REQ := wire#w1, PORT := "Local~CM_1241_(RS232)_1", BUFFER := "DELTA D"."MIN F0", LENGTH :=, PTRCL :=, DONE =>, ERROR =>, STATUS =>)
   END_RUNG
   RUNG wire#powerrail
      Contact( "CLOSURE ON" )
      { S7_Templates := "SrcType := Int" } EQ_Contact(in1 := "IEC_Counter_0_DB_5".CV, in2 := 6)
      { S7_Templates := "time_type := Time" } "IEC_Timer_0_DB_128".TON(pt := T#200MS, et =>)
      P_Trig( "PP5" )
   END_RUNG wire#w1
   // the same network as SCL:
   "IEC_Timer_0_DB_128".TON(IN := "CLOSURE ON" AND ("IEC_Counter_0_DB_5".CV = 6), PT := T#200MS);
   #_w1 := "IEC_Timer_0_DB_128".Q AND NOT "PP5";   // rising edge
   "PP5" := "IEC_Timer_0_DB_128".Q;
   IF "AlwaysTRUE" THEN
       "SEND_PTP_DB_36"(REQ := #_w1, PORT := "Local~CM_1241_(RS232)_1", BUFFER := "DELTA D"."MIN F0");   // SEND_PTP
   END_IF;
END_REGION

REGION Network 17
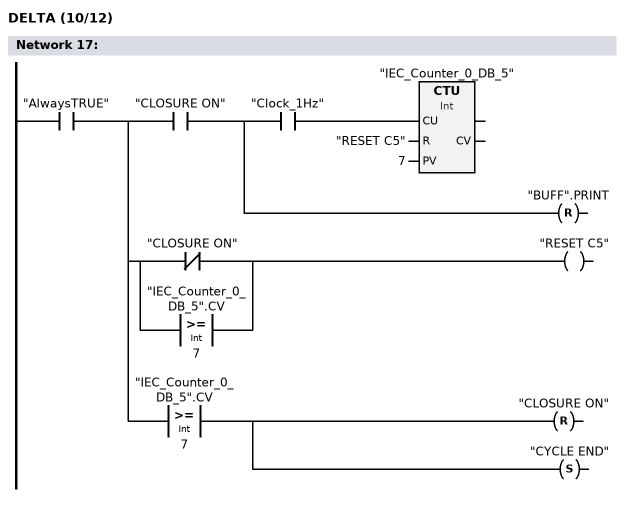
   RUNG wire#powerrail
      Contact( "AlwaysTRUE" )
      wire#w1
      Contact( "CLOSURE ON" )
      wire#w2
      Contact( "Clock_1Hz" )
      { S7_Templates := "value_type := Int" } "IEC_Counter_0_DB_5".CTU(r := "RESET C5", pv := 7, cv =>)
   END_RUNG
   RUNG wire#w2
      R_Coil( "BUFF".PRINT )
   END_RUNG
   RUNG wire#w1
      I_Contact( "CLOSURE ON" )
      wire#w3
      Coil( "RESET C5" )
   END_RUNG
   RUNG wire#w1
      { S7_Templates := "SrcType := Int" } GE_Contact(in1 := "IEC_Counter_0_DB_5".CV, in2 := 7)
   END_RUNG wire#w3
   RUNG wire#w1
      { S7_Templates := "SrcType := Int" } GE_Contact(in1 := "IEC_Counter_0_DB_5".CV, in2 := 7)
      wire#w4
      R_Coil( "CLOSURE ON" )
   END_RUNG
   RUNG wire#w4
      S_Coil( "CYCLE END" )
   END_RUNG
   // the same network as SCL:
   #_w1 := "AlwaysTRUE" AND "CLOSURE ON";
   "IEC_Counter_0_DB_5".CTU(CU := #_w1 AND "Clock_1Hz", R := "RESET C5", PV := 7);
   IF #_w1 THEN "BUFF".PRINT := FALSE; END_IF;
   "RESET C5" := "AlwaysTRUE" AND (NOT "CLOSURE ON" OR ("IEC_Counter_0_DB_5".CV >= 7));
   IF "AlwaysTRUE" AND ("IEC_Counter_0_DB_5".CV >= 7) THEN
       "CLOSURE ON" := FALSE;
       "CYCLE END" := TRUE;
   END_IF;
END_REGION

REGION Network 18
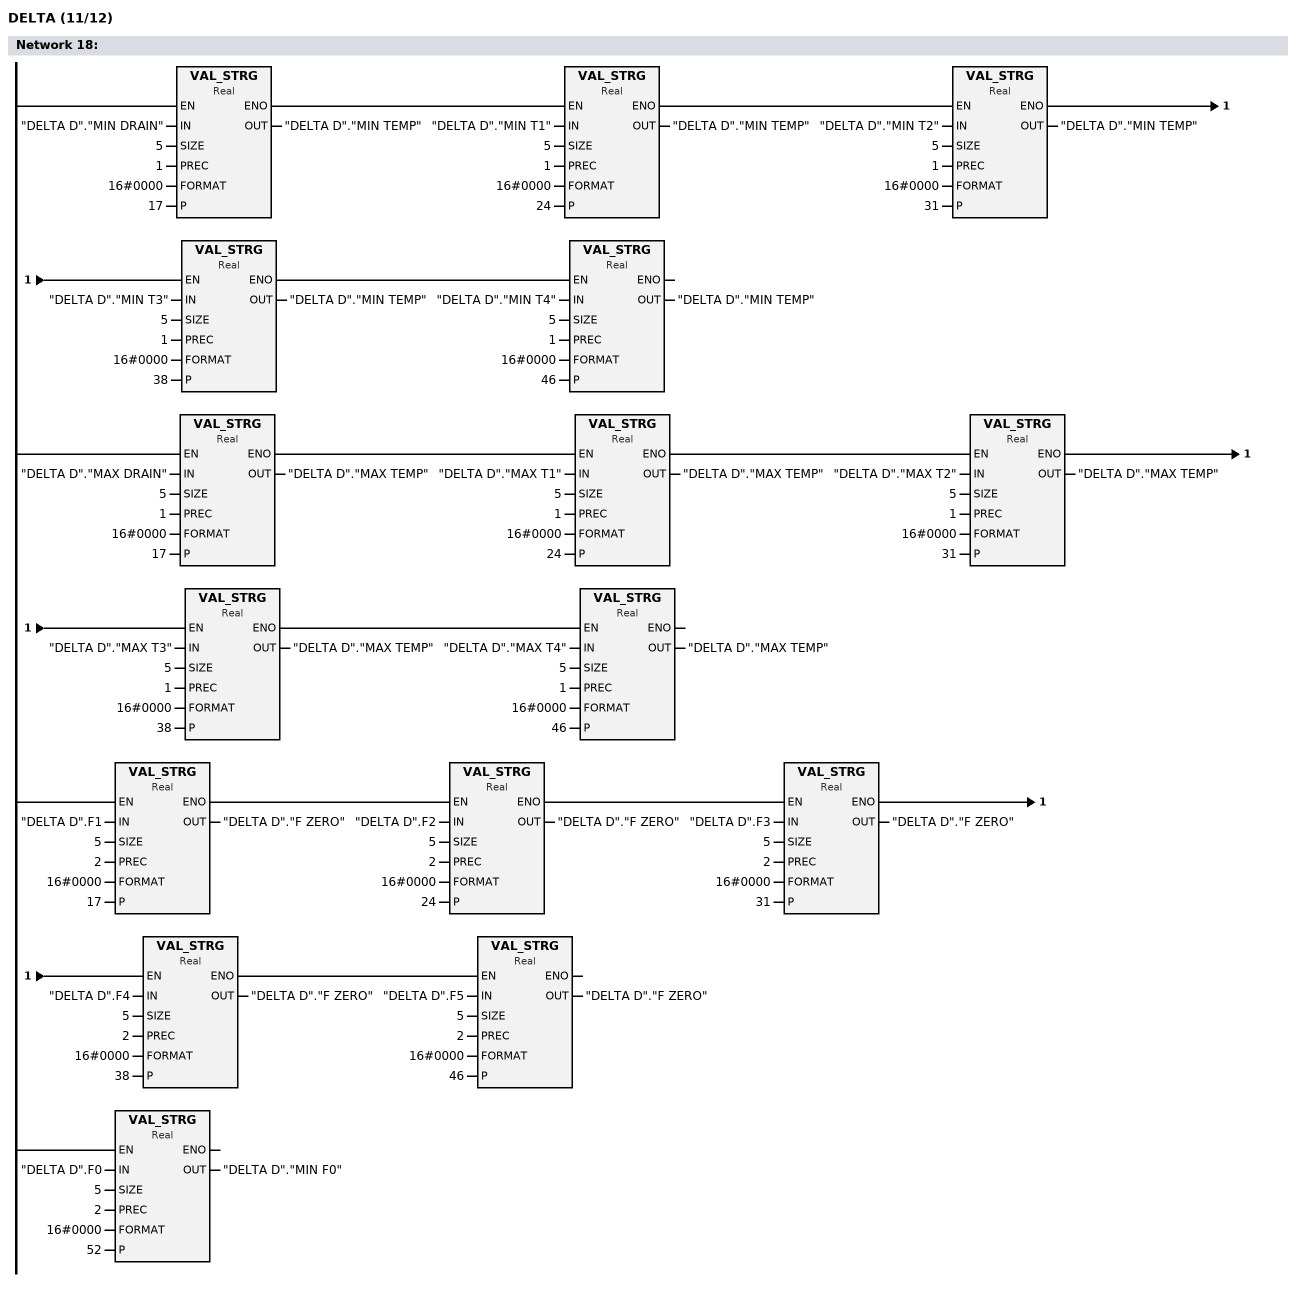
   RUNG wire#powerrail
      { S7_Templates := "[value_type := Real, str_type := String]" } VAL_STRG(IN := "DELTA D"."MIN DRAIN", SIZE := 5, PREC := 1, FORMAT := 16#0000, P := 17, OUT => "DELTA D"."MIN TEMP")
      { S7_Templates := "[value_type := Real, str_type := String]" } VAL_STRG(IN := "DELTA D"."MIN T1", SIZE := 5, PREC := 1, FORMAT := 16#0000, P := 24, OUT => "DELTA D"."MIN TEMP")
      { S7_Templates := "[value_type := Real, str_type := String]" } VAL_STRG(IN := "DELTA D"."MIN T2", SIZE := 5, PREC := 1, FORMAT := 16#0000, P := 31, OUT => "DELTA D"."MIN TEMP")
      { S7_Templates := "[value_type := Real, str_type := String]" } VAL_STRG(IN := "DELTA D"."MIN T3", SIZE := 5, PREC := 1, FORMAT := 16#0000, P := 38, OUT => "DELTA D"."MIN TEMP")
      { S7_Templates := "[value_type := Real, str_type := String]" } VAL_STRG(IN := "DELTA D"."MIN T4", SIZE := 5, PREC := 1, FORMAT := 16#0000, P := 46, OUT => "DELTA D"."MIN TEMP")
   END_RUNG
   RUNG wire#powerrail
      { S7_Templates := "[value_type := Real, str_type := String]" } VAL_STRG(IN := "DELTA D"."MAX DRAIN", SIZE := 5, PREC := 1, FORMAT := 16#0000, P := 17, OUT => "DELTA D"."MAX TEMP")
      { S7_Templates := "[value_type := Real, str_type := String]" } VAL_STRG(IN := "DELTA D"."MAX T1", SIZE := 5, PREC := 1, FORMAT := 16#0000, P := 24, OUT => "DELTA D"."MAX TEMP")
      { S7_Templates := "[value_type := Real, str_type := String]" } VAL_STRG(IN := "DELTA D"."MAX T2", SIZE := 5, PREC := 1, FORMAT := 16#0000, P := 31, OUT => "DELTA D"."MAX TEMP")
      { S7_Templates := "[value_type := Real, str_type := String]" } VAL_STRG(IN := "DELTA D"."MAX T3", SIZE := 5, PREC := 1, FORMAT := 16#0000, P := 38, OUT => "DELTA D"."MAX TEMP")
      { S7_Templates := "[value_type := Real, str_type := String]" } VAL_STRG(IN := "DELTA D"."MAX T4", SIZE := 5, PREC := 1, FORMAT := 16#0000, P := 46, OUT => "DELTA D"."MAX TEMP")
   END_RUNG
   RUNG wire#powerrail
      { S7_Templates := "[value_type := Real, str_type := String]" } VAL_STRG(IN := "DELTA D".F1, SIZE := 5, PREC := 2, FORMAT := 16#0000, P := 17, OUT => "DELTA D"."F ZERO")
      { S7_Templates := "[value_type := Real, str_type := String]" } VAL_STRG(IN := "DELTA D".F2, SIZE := 5, PREC := 2, FORMAT := 16#0000, P := 24, OUT => "DELTA D"."F ZERO")
      { S7_Templates := "[value_type := Real, str_type := String]" } VAL_STRG(IN := "DELTA D".F3, SIZE := 5, PREC := 2, FORMAT := 16#0000, P := 31, OUT => "DELTA D"."F ZERO")
      { S7_Templates := "[value_type := Real, str_type := String]" } VAL_STRG(IN := "DELTA D".F4, SIZE := 5, PREC := 2, FORMAT := 16#0000, P := 38, OUT => "DELTA D"."F ZERO")
      { S7_Templates := "[value_type := Real, str_type := String]" } VAL_STRG(IN := "DELTA D".F5, SIZE := 5, PREC := 2, FORMAT := 16#0000, P := 46, OUT => "DELTA D"."F ZERO")
   END_RUNG
   RUNG wire#powerrail
      { S7_Templates := "[value_type := Real, str_type := String]" } VAL_STRG(IN := "DELTA D".F0, SIZE := 5, PREC := 2, FORMAT := 16#0000, P := 52, OUT => "DELTA D"."MIN F0")
   END_RUNG
   // the same network as SCL:
   VAL_STRG(IN := "DELTA D"."MIN DRAIN",
            SIZE := 5,
            PREC := 1,
            FORMAT := 16#0000,
            P := 17,
            OUT => "DELTA D"."MIN TEMP",
            ENO => #_w1);
   VAL_STRG(EN := #_w1,
            IN := "DELTA D"."MIN T1",
            SIZE := 5,
            PREC := 1,
            FORMAT := 16#0000,
            P := 24,
            OUT => "DELTA D"."MIN TEMP",
            ENO => #_w2);
   VAL_STRG(EN := #_w2,
            IN := "DELTA D"."MIN T2",
            SIZE := 5,
            PREC := 1,
            FORMAT := 16#0000,
            P := 31,
            OUT => "DELTA D"."MIN TEMP",
            ENO => #_w3);
   VAL_STRG(EN := #_w3,
            IN := "DELTA D"."MIN T3",
            SIZE := 5,
            PREC := 1,
            FORMAT := 16#0000,
            P := 38,
            OUT => "DELTA D"."MIN TEMP",
            ENO => #_w4);
   IF #_w4 THEN
       VAL_STRG(IN := "DELTA D"."MIN T4",
                SIZE := 5,
                PREC := 1,
                FORMAT := 16#0000,
                P := 46,
                OUT => "DELTA D"."MIN TEMP");
   END_IF;
   VAL_STRG(IN := "DELTA D"."MAX DRAIN",
            SIZE := 5,
            PREC := 1,
            FORMAT := 16#0000,
            P := 17,
            OUT => "DELTA D"."MAX TEMP",
            ENO => #_w5);
   VAL_STRG(EN := #_w5,
            IN := "DELTA D"."MAX T1",
            SIZE := 5,
            PREC := 1,
            FORMAT := 16#0000,
            P := 24,
            OUT => "DELTA D"."MAX TEMP",
            ENO => #_w6);
   VAL_STRG(EN := #_w6,
            IN := "DELTA D"."MAX T2",
            SIZE := 5,
            PREC := 1,
            FORMAT := 16#0000,
            P := 31,
            OUT => "DELTA D"."MAX TEMP",
            ENO => #_w7);
   VAL_STRG(EN := #_w7,
            IN := "DELTA D"."MAX T3",
            SIZE := 5,
            PREC := 1,
            FORMAT := 16#0000,
            P := 38,
            OUT => "DELTA D"."MAX TEMP",
            ENO => #_w8);
   IF #_w8 THEN
       VAL_STRG(IN := "DELTA D"."MAX T4",
                SIZE := 5,
                PREC := 1,
                FORMAT := 16#0000,
                P := 46,
                OUT => "DELTA D"."MAX TEMP");
   END_IF;
   VAL_STRG(IN := "DELTA D".F1,
            SIZE := 5,
            PREC := 2,
            FORMAT := 16#0000,
            P := 17,
            OUT => "DELTA D"."F ZERO",
            ENO => #_w9);
   VAL_STRG(EN := #_w9,
            IN := "DELTA D".F2,
            SIZE := 5,
            PREC := 2,
            FORMAT := 16#0000,
            P := 24,
            OUT => "DELTA D"."F ZERO",
            ENO => #_w10);
   VAL_STRG(EN := #_w10,
            IN := "DELTA D".F3,
            SIZE := 5,
            PREC := 2,
            FORMAT := 16#0000,
            P := 31,
            OUT => "DELTA D"."F ZERO",
            ENO => #_w11);
   VAL_STRG(EN := #_w11,
            IN := "DELTA D".F4,
            SIZE := 5,
            PREC := 2,
            FORMAT := 16#0000,
            P := 38,
            OUT => "DELTA D"."F ZERO",
            ENO => #_w12);
   IF #_w12 THEN
       VAL_STRG(IN := "DELTA D".F5, SIZE := 5, PREC := 2, FORMAT := 16#0000, P := 46, OUT => "DELTA D"."F ZERO");
   END_IF;
   VAL_STRG(IN := "DELTA D".F0, SIZE := 5, PREC := 2, FORMAT := 16#0000, P := 52, OUT => "DELTA D"."MIN F0");
END_REGION

REGION Network 19
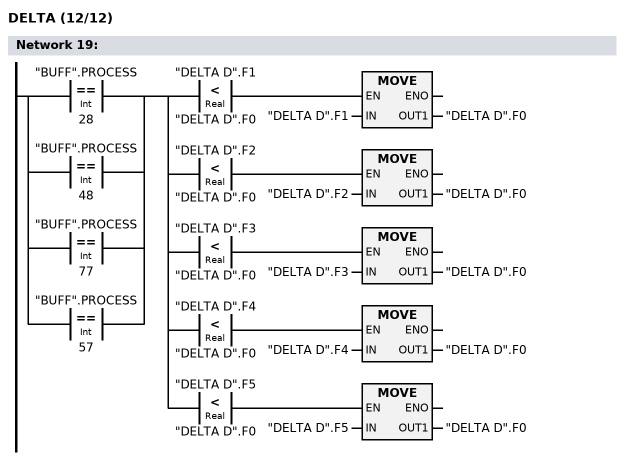
   RUNG wire#powerrail
      { S7_Templates := "SrcType := Int" } EQ_Contact(in1 := "BUFF".PROCESS, in2 := 28)
      wire#w1
      { S7_Templates := "SrcType := Real" } LT_Contact(in1 := "DELTA D".F1, in2 := "DELTA D".F0)
      Move(in := "DELTA D".F1, out1 => "DELTA D".F0)
   END_RUNG
   RUNG wire#powerrail
      { S7_Templates := "SrcType := Int" } EQ_Contact(in1 := "BUFF".PROCESS, in2 := 48)
   END_RUNG wire#w1
   RUNG wire#powerrail
      { S7_Templates := "SrcType := Int" } EQ_Contact(in1 := "BUFF".PROCESS, in2 := 77)
   END_RUNG wire#w1
   RUNG wire#powerrail
      { S7_Templates := "SrcType := Int" } EQ_Contact(in1 := "BUFF".PROCESS, in2 := 57)
   END_RUNG wire#w1
   RUNG wire#w1
      { S7_Templates := "SrcType := Real" } LT_Contact(in1 := "DELTA D".F2, in2 := "DELTA D".F0)
      Move(in := "DELTA D".F2, out1 => "DELTA D".F0)
   END_RUNG
   RUNG wire#w1
      { S7_Templates := "SrcType := Real" } LT_Contact(in1 := "DELTA D".F3, in2 := "DELTA D".F0)
      Move(in := "DELTA D".F3, out1 => "DELTA D".F0)
   END_RUNG
   RUNG wire#w1
      { S7_Templates := "SrcType := Real" } LT_Contact(in1 := "DELTA D".F4, in2 := "DELTA D".F0)
      Move(in := "DELTA D".F4, out1 => "DELTA D".F0)
   END_RUNG
   RUNG wire#w1
      { S7_Templates := "SrcType := Real" } LT_Contact(in1 := "DELTA D".F5, in2 := "DELTA D".F0)
      Move(in := "DELTA D".F5, out1 => "DELTA D".F0)
   END_RUNG
   // the same network as SCL:
   #_w1 := ("BUFF".PROCESS = 28) OR ("BUFF".PROCESS = 48) OR ("BUFF".PROCESS = 77) OR ("BUFF".PROCESS = 57);
   IF #_w1 AND ("DELTA D".F1 < "DELTA D".F0) THEN "DELTA D".F0 := "DELTA D".F1; END_IF;
   IF #_w1 AND ("DELTA D".F2 < "DELTA D".F0) THEN "DELTA D".F0 := "DELTA D".F2; END_IF;
   IF #_w1 AND ("DELTA D".F3 < "DELTA D".F0) THEN "DELTA D".F0 := "DELTA D".F3; END_IF;
   IF #_w1 AND ("DELTA D".F4 < "DELTA D".F0) THEN "DELTA D".F0 := "DELTA D".F4; END_IF;
   IF #_w1 AND ("DELTA D".F5 < "DELTA D".F0) THEN "DELTA D".F0 := "DELTA D".F5; END_IF;
END_REGION
END_FUNCTION
